INTERFACE I_MotionAxisHome

END_INTERFACE

(* stored: Version 1.1.0.1
   Itf I_MotionAxisHome: Id {9a574bd6-8158-416c-bf7f-7449d94d0592} *)
